Omron CX-Programmer project NewProject (CX-Programmer 9.61)

# PLC NewPLC1: CP1E N30

## Global symbols (name address type ; comment)
0 CHANNEL  ; CJP
0.00 BOOL  ; ON
0.01 BOOL  ; OFF
0.02 BOOL  ; JMP TRIGGER
100.00 BOOL  ; LAMP
100.01 BOOL  ; LAMP2
200.00 BOOL  ; K1

## Program NewProgram1 (cyclic task 0)

### Section Section1

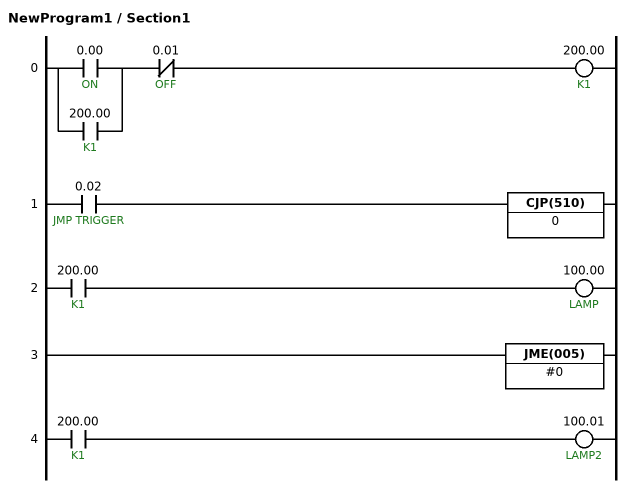
; rung 0
LD 0.00  ; ON
OR 200.00  ; K1
ANDNOT 0.01  ; OFF
OUT 200.00  ; K1
; rung 1
LD 0.02  ; JMP TRIGGER
CJP(510) 0
; rung 2
LD 200.00  ; K1
OUT 100.00  ; LAMP
; rung 3
JME(005) #0
; rung 4
LD 200.00  ; K1
OUT 100.01  ; LAMP2

### Section END
; rung 0
END(001)